(* IEC 61131-3 sources: Projeto_Automacao_Arduino/Projeto_AI/build, 2 files *)

(* ---- plc.st ---- *)
TYPE
  LOGLEVEL : (CRITICAL, WARNING, INFO, DEBUG) := INFO;
END_TYPE

FUNCTION_BLOCK LOGGER
  VAR_INPUT
    TRIG : BOOL;
    MSG : STRING;
    LEVEL : LOGLEVEL := INFO;
  END_VAR
  VAR
    TRIG0 : BOOL;
  END_VAR

  IF TRIG AND NOT TRIG0 THEN
  {{
   LogMessage(GetFbVar(LEVEL),(char*)GetFbVar(MSG, .body),GetFbVar(MSG, .len));
  }}
  END_IF;
  TRIG0:=TRIG;
END_FUNCTION_BLOCK

FUNCTION_BLOCK python_eval
  VAR_INPUT
    TRIG : BOOL;
    CODE : STRING;
  END_VAR
  VAR_OUTPUT
    ACK : BOOL;
    RESULT : STRING;
  END_VAR
  VAR
    STATE : DWORD;
    BUFFER : STRING;
    PREBUFFER : STRING;
    TRIGM1 : BOOL;
    TRIGGED : BOOL;
  END_VAR

  {extern void __PythonEvalFB(int, PYTHON_EVAL*);__PythonEvalFB(0, data__);}
END_FUNCTION_BLOCK

FUNCTION_BLOCK python_poll
  VAR_INPUT
    TRIG : BOOL;
    CODE : STRING;
  END_VAR
  VAR_OUTPUT
    ACK : BOOL;
    RESULT : STRING;
  END_VAR
  VAR
    STATE : DWORD;
    BUFFER : STRING;
    PREBUFFER : STRING;
    TRIGM1 : BOOL;
    TRIGGED : BOOL;
  END_VAR

  {extern void __PythonEvalFB(int, PYTHON_EVAL*);__PythonEvalFB(1,(PYTHON_EVAL*)(void*)data__);}
END_FUNCTION_BLOCK

FUNCTION_BLOCK python_gear
  VAR_INPUT
    N : UINT;
    TRIG : BOOL;
    CODE : STRING;
  END_VAR
  VAR_OUTPUT
    ACK : BOOL;
    RESULT : STRING;
  END_VAR
  VAR
    py_eval : python_eval;
    COUNTER : UINT;
    ADD10_OUT : UINT;
    EQ13_OUT : BOOL;
    SEL15_OUT : UINT;
    AND7_OUT : BOOL;
  END_VAR

  ADD10_OUT := ADD(COUNTER, 1);
  EQ13_OUT := EQ(N, ADD10_OUT);
  SEL15_OUT := SEL(EQ13_OUT, ADD10_OUT, 0);
  COUNTER := SEL15_OUT;
  AND7_OUT := AND(EQ13_OUT, TRIG);
  py_eval(TRIG := AND7_OUT, CODE := CODE);
  ACK := py_eval.ACK;
  RESULT := py_eval.RESULT;
END_FUNCTION_BLOCK

PROGRAM Controle_Servo
  VAR
    START : BOOL;
    STOP : BOOL;
    CONTROL : BOOL;
    START_LED : BOOL;
    STOP_LED : BOOL := True;
    OUTPUT : BOOL;
  END_VAR
  VAR
    TON0 : TON;
  END_VAR
  VAR
    ENABLE_CONTROL : BOOL;
  END_VAR

  START_LED := NOT(STOP) AND (START OR START_LED);
  IF NOT(STOP) AND (START OR START_LED) THEN
    ENABLE_CONTROL := TRUE; (*set*)
  END_IF;
  STOP_LED := NOT(START) AND (STOP OR STOP_LED);
  IF NOT(START) AND (STOP OR STOP_LED) THEN
    ENABLE_CONTROL := FALSE; (*reset*)
  END_IF;
  IF NOT(START) AND (STOP OR STOP_LED) THEN
    OUTPUT := FALSE; (*reset*)
  END_IF;
  IF CONTROL AND ENABLE_CONTROL THEN
    OUTPUT := TRUE; (*set*)
  END_IF;
  TON0(IN := OUTPUT, PT := T#5s);
  IF TON0.Q THEN
    OUTPUT := FALSE; (*reset*)
  END_IF;
END_PROGRAM

CONFIGURATION Config0

  RESOURCE Res0 ON PLC
    TASK task0(INTERVAL := T#20ms,PRIORITY := 0);
    PROGRAM instance0 WITH task0 : Controle_Servo;
  END_RESOURCE
END_CONFIGURATION

(* ---- generated_plc.st ---- *)
PROGRAM Controle_Servo
  VAR
    START AT %IX100.0 : BOOL;
    STOP AT %IX100.1 : BOOL;
    CONTROL AT %IX100.2 : BOOL;
    START_LED AT %QX100.0 : BOOL;
    STOP_LED AT %QX100.1 : BOOL := True;
    OUTPUT AT %QX100.2 : BOOL;
  END_VAR
  VAR
    TON0 : TON;
  END_VAR
  VAR
    ENABLE_CONTROL AT %MX100 : BOOL;
  END_VAR

  START_LED := NOT(STOP) AND (START OR START_LED);
  IF NOT(STOP) AND (START OR START_LED) THEN
    ENABLE_CONTROL := TRUE; (*set*)
  END_IF;
  STOP_LED := NOT(START) AND (STOP OR STOP_LED);
  IF NOT(START) AND (STOP OR STOP_LED) THEN
    ENABLE_CONTROL := FALSE; (*reset*)
  END_IF;
  IF NOT(START) AND (STOP OR STOP_LED) THEN
    OUTPUT := FALSE; (*reset*)
  END_IF;
  IF CONTROL AND ENABLE_CONTROL THEN
    OUTPUT := TRUE; (*set*)
  END_IF;
  TON0(IN := OUTPUT, PT := T#5s);
  IF TON0.Q THEN
    OUTPUT := FALSE; (*reset*)
  END_IF;
END_PROGRAM

CONFIGURATION Config0

  RESOURCE Res0 ON PLC
    TASK task0(INTERVAL := T#20ms,PRIORITY := 0);
    PROGRAM instance0 WITH task0 : Controle_Servo;
  END_RESOURCE
END_CONFIGURATION
